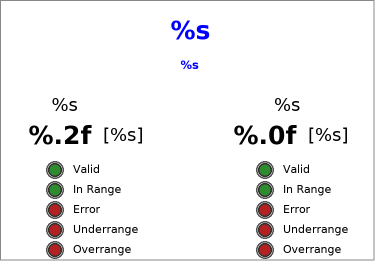
VISUALIZATION GUI_TEMPLATE_SBG232  // 375x261
VAR_IN_OUT
	m_Instance:	FB_CRYO_SBG232;
END_VAR
    Rectangle (41,10 299x40), "%s", tooltip "Sensor Name", text variable: m_Instance.stat.sName
    Rectangle (20,120 80x30), "%.2f", text variable: m_Instance.stat.flow.lrValue
    Rectangle (30,90 70x30), "%s", text variable: m_Instance.stat.flow.sType
    Rectangle (100,120 70x30), "[%s]", text variable: m_Instance.stat.flow.sUnits
    Rectangle (225,120 80x30), "%.0f", text variable: m_Instance.stat.temp.lrValue
    Rectangle (220,90 135x30), "%s", text variable: m_Instance.stat.temp.sType
    Rectangle (305,120 70x30), "[%s]", text variable: m_Instance.stat.temp.sUnits
    Lamp1 (45,160 20x20), tooltip "If ON, reading is valid.", variable: m_Instance.stat.flow.bValid, style: Lamp-Lamp1-Green
    Lamp1 (45,180 20x20), tooltip "If ON, reading is in expected range.", variable: m_Instance.stat.flow.bInRange, style: Lamp-Lamp1-Green
    Rectangle (5,50 370x30), "%s", tooltip "Sensor Status", text variable: m_Instance.stat.sStatus
    Lamp1 (45,220 20x20), tooltip "If ON, reading is in underrange.", variable: m_Instance.stat.flow.bUnderrange, style: Lamp-Lamp1-Red
    Lamp1 (45,240 20x20), tooltip "If ON, reading is in overrange.", variable: m_Instance.stat.flow.bOverrange, style: Lamp-Lamp1-Red
    Lamp1 (45,200 20x20), tooltip "If ON, reading is in error.", variable: m_Instance.stat.flow.bError, style: Lamp-Lamp1-Red
    Label (70,158 87x23), "Valid"
    Label (70,178 87x23), "In Range"
    Label (70,198 87x23), "Error"
    Label (70,218 87x23), "Underrange"
    Label (70,238 87x23), "Overrange"
    Lamp1 (255,160 20x20), tooltip "If ON, reading is valid.", variable: m_Instance.stat.temp.bValid, style: Lamp-Lamp1-Green
    Lamp1 (255,180 20x20), tooltip "If ON, reading is in expected range.", variable: m_Instance.stat.temp.bInRange, style: Lamp-Lamp1-Green
    Lamp1 (255,220 20x20), tooltip "If ON, reading is in underrange.", variable: m_Instance.stat.temp.bUnderrange, style: Lamp-Lamp1-Red
    Lamp1 (255,240 20x20), tooltip "If ON, reading is in overrange.", variable: m_Instance.stat.temp.bOverrange, style: Lamp-Lamp1-Red
    Lamp1 (255,200 20x20), tooltip "If ON, reading is in error.", variable: m_Instance.stat.temp.bError, style: Lamp-Lamp1-Red
    Label (280,158 87x23), "Valid"
    Label (280,178 87x23), "In Range"
    Label (280,198 87x23), "Error"
    Label (280,218 87x23), "Underrange"
    Label (280,238 87x23), "Overrange"
END_VISUALIZATION

(* stored: Version 1.1.0.1, ProductVersion 3.1.4024.12
   Visu GUI_TEMPLATE_SBG232: Id {1a0cb542-d5ee-4483-8edc-60d6cfc84a9d} *)
